// TIA Portal V16 export
// export: Created 2020-12-17T10:21:39.4735782Z, ExportSetting WithDefaults, DisplayName Totally Integrated Automation Portal, DisplayVersion V16 Update 2, DisplayName TIA Portal Version Control Interface, DisplayVersion V16 Update 2, DisplayName TIA Portal Openness, DisplayVersion V16 Update 2, DisplayName STEP 7 Professional, DisplayVersion V16 Update 2, DisplayName STEP 7 Safety, DisplayVersion V16, DisplayName WinCC Advanced / Unified PC, DisplayVersion V16 Update 2
FUNCTION "Block_F1" : Bool   // FC2, FBD
TITLE = XOR function
{ S7_Optimized_Access := 'TRUE' }
VERSION : 0.1
// As an example
// stored: AutoNumber true, IsIECCheckEnabled false, SetENOAutomatically false, UDAEnableTagReadback false
   VAR_INPUT
      Arg1 : Bool;
      Arg2 : Bool;
   END_VAR
BEGIN

REGION Network 1: N1
   // Body
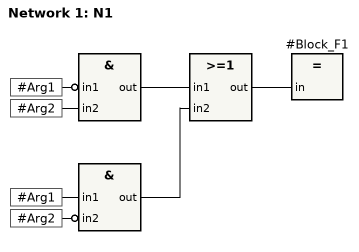
   #Block_F1 := (NOT #Arg1 AND #Arg2) OR (#Arg1 AND NOT #Arg2);
END_REGION
END_FUNCTION
